(* IEC 61131-3 sources: MotionTestBenchMaster/Logical/02_HMI/0210_PAR/PAR, 10 files *)

(* ---- HMI_PAC_1.st ---- *)
(*HMI_PAC_1 Initialization Action for Filler PLC*)
(*Author = UTERF*)
(*DB Version : 0.11*)
(*File Version : 2.88*)

ACTION HMI_PAC_1_Init :
        HMI_PAC_1._000 := 0;
        HMI_PAC_1._001 := 20;
        HMI_PAC_1._002 := 200;
        HMI_PAC_1._003 := 0;
        HMI_PAC_1._004 := 1;
        HMI_PAC_1._005 := 1;
        HMI_PAC_1._006 := 1;
        HMI_PAC_1._007 := 210;
        HMI_PAC_1._008 := 105;
        HMI_PAC_1._009 := 0;
        HMI_PAC_1._013 := 205;
        HMI_PAC_1._014 := 0;
        HMI_PAC_1._016 := 0;
        HMI_PAC_1._017 := 0;
        HMI_PAC_1._018 := 0;
        HMI_PAC_1._019 := 89;
        HMI_PAC_1._020 := 118;
        HMI_PAC_1._021 := 0;
        HMI_PAC_1._022 := 0;
        HMI_PAC_1._023 := 0;
        HMI_PAC_1._024 := 0;
        HMI_PAC_1._045 := 0;
        HMI_PAC_1._070 := 0;
        HMI_PAC_1._071 := 0;
        HMI_PAC_1._100 := 91;
        HMI_PAC_1._101 := 75;
        HMI_PAC_1._102 := 5;
        HMI_PAC_1._103 := 0;
        HMI_PAC_1._104 := 85;
        HMI_PAC_1._105 := 0;
        HMI_PAC_1._106 := 0;
        HMI_PAC_1._107 := 0;
        HMI_PAC_1._108 := 0;
        HMI_PAC_1._110 := 0;
        HMI_PAC_1._111 := 0;
        HMI_PAC_1._112 := 0;
        HMI_PAC_1._113 := 0;
        HMI_PAC_1._114 := 0;
        HMI_PAC_1._115 := 0;
        HMI_PAC_1._117 := 0;
        HMI_PAC_1._118 := 0;
        HMI_PAC_1._120 := 0;
        HMI_PAC_1._121 := 0;
        HMI_PAC_1._122 := 0;
        HMI_PAC_1._123 := 0;
        HMI_PAC_1._124 := 0;
        HMI_PAC_1._125 := 0;
        HMI_PAC_1._126 := 0;
        HMI_PAC_1._127 := 0;
        HMI_PAC_1._128 := 0;
        HMI_PAC_1._129 := 1;
        HMI_PAC_1._130 := 33;
        HMI_PAC_1._131 := 1;
        HMI_PAC_1._132 := 0;
        HMI_PAC_1._133 := 1;
        HMI_PAC_1._134 := 1;
        HMI_PAC_1._145 := 0;
        HMI_PAC_1._146 := 0;
        HMI_PAC_1._150 := 6;
        HMI_PAC_1._151 := 1;
        HMI_PAC_1._152 := 74;
        HMI_PAC_1._200 := 0;
        HMI_PAC_1._201 := 0;
        HMI_PAC_1._202 := 0;
        HMI_PAC_1._203 := 0;
        HMI_PAC_1._204 := 0;
        HMI_PAC_1._205 := 0;
        HMI_PAC_1._206 := 0;
        HMI_PAC_1._207 := 0;
        HMI_PAC_1._208 := 0;
        HMI_PAC_1._209 := 0;
        HMI_PAC_1._210 := 0;
        HMI_PAC_1._211 := 0;
        HMI_PAC_1._212 := 0;
        HMI_PAC_1._213 := 0;
        HMI_PAC_1._214 := 0;
        HMI_PAC_1._215 := 0;
        HMI_PAC_1._219 := 0;
        HMI_PAC_1._220 := 0;
        HMI_PAC_1._245 := 0;
        HMI_PAC_1._246 := 0;
        HMI_PAC_1._300 := 0;
        HMI_PAC_1._301 := 0;
        HMI_PAC_1._302 := 0;
        HMI_PAC_1._303 := 0;
        HMI_PAC_1._304 := 0;
        HMI_PAC_1._305 := 0;
        HMI_PAC_1._306 := 0;
        HMI_PAC_1._307 := 0;
        HMI_PAC_1._400 := 0;
        HMI_PAC_1._401 := 0;
        HMI_PAC_1._402 := 0;
        HMI_PAC_1._403 := 0;
        HMI_PAC_1._404 := 0;
        HMI_PAC_1._405 := 0;
        HMI_PAC_1._406 := 0;
        HMI_PAC_1._407 := 0;
        HMI_PAC_1._408 := 0;
        HMI_PAC_1._409 := 0;
        HMI_PAC_1._410 := 0;
        HMI_PAC_1._411 := 0;
        HMI_PAC_1._412 := 0;
        HMI_PAC_1._413 := 0;
        HMI_PAC_1._415 := 0;
        HMI_PAC_1._416 := 0;
        HMI_PAC_1._417 := 0;
        HMI_PAC_1._418 := 0;
        HMI_PAC_1._419 := 0;
        HMI_PAC_1._420 := 0;
        HMI_PAC_1._422 := 0;
        HMI_PAC_1._423 := 0;
        HMI_PAC_1._500 := 0;
        HMI_PAC_1._501 := 0;
        HMI_PAC_1._502 := 0;
        HMI_PAC_1._503 := 0;
        HMI_PAC_1._504 := 0;
        HMI_PAC_1._510 := 0;
        HMI_PAC_1._600 := 0;
        HMI_PAC_1._601 := 0;
        HMI_PAC_1._605 := 0;
        HMI_PAC_1._606 := 0;
        HMI_PAC_1._610 := 0;
        HMI_PAC_1._700 := 0;
        HMI_PAC_1._701 := 0;
        HMI_PAC_1._702 := 0;
        HMI_PAC_1._703 := 0;
        HMI_PAC_1._704 := 1;
        HMI_PAC_1._705 := 1;
        HMI_PAC_1._706 := 1;
        HMI_PAC_1._800 := 0;
END_ACTION

(* ---- HMI_PAM_1.st ---- *)
(*HMI_PAM_1 Initialization Action for Filler PLC*)
(*Author = ????*)
(*DB Version : 0.10*)
(*File Version : 2.88*)

ACTION HMI_PAM_1_Init :
        HMI_PAM_1._000 := 50;
        HMI_PAM_1._001 := 20000;
        HMI_PAM_1._002 := 60;
        HMI_PAM_1._003 := 5000;
        HMI_PAM_1._004 := 8000;
        HMI_PAM_1._005 := 5000;
        HMI_PAM_1._006 := 25000;
        HMI_PAM_1._007 := 15000;
        HMI_PAM_1._008 := 20000;
        HMI_PAM_1._009 := 20000;
        HMI_PAM_1._010 := 1500;
        HMI_PAM_1._011 := 8;
        HMI_PAM_1._012 := 8;
        HMI_PAM_1._013 := 0.13;
        HMI_PAM_1._014 := 20000;
        HMI_PAM_1._015 := 20000;
        HMI_PAM_1._020 := 55200;
        HMI_PAM_1._021 := 400;
        HMI_PAM_1._022 := 2;
        HMI_PAM_1._023 := 600;
        HMI_PAM_1._030 := 300;
        HMI_PAM_1._031 := 2;
        HMI_PAM_1._032 := 2;
        HMI_PAM_1._036 := 0;
        HMI_PAM_1._040 := 300;
        HMI_PAM_1._041 := 5;
        HMI_PAM_1._044 := 0;
        HMI_PAM_1._045 := 0;
        HMI_PAM_1._046 := 0;
        HMI_PAM_1._047 := 0;
        HMI_PAM_1._048 := 10;
        HMI_PAM_1._049 := 1;
        HMI_PAM_1._050 := 60;
        HMI_PAM_1._051 := 0;
        HMI_PAM_1._052 := 0;
        HMI_PAM_1._053 := 0;
        HMI_PAM_1._054 := 0;
        HMI_PAM_1._055 := 10000;
        HMI_PAM_1._056 := 20000;
        HMI_PAM_1._057 := 0;
        HMI_PAM_1._058 := 0;
        HMI_PAM_1._060 := 5;
        HMI_PAM_1._061 := 100;
        HMI_PAM_1._065 := 50;
        HMI_PAM_1._080 := 0;
        HMI_PAM_1._081 := 0;
        HMI_PAM_1._082 := 0;
        HMI_PAM_1._083 := 0;
        HMI_PAM_1._084 := 0;
        HMI_PAM_1._085 := 0;
        HMI_PAM_1._086 := 3;
        HMI_PAM_1._087 := 3;
        HMI_PAM_1._088 := 3;
        HMI_PAM_1._089 := 3;
        HMI_PAM_1._090 := 1000000;
        HMI_PAM_1._091 := 40000;
        HMI_PAM_1._092 := 3.2;
        HMI_PAM_1._093 := 3.2;
        HMI_PAM_1._100 := 0;
        HMI_PAM_1._101 := 0;
        HMI_PAM_1._102 := 0;
        HMI_PAM_1._103 := 100;
        HMI_PAM_1._104 := 100;
        HMI_PAM_1._105 := 2;
        HMI_PAM_1._106 := 15;
        HMI_PAM_1._107 := 10;
        HMI_PAM_1._108 := 5;
        HMI_PAM_1._109 := 5;
        HMI_PAM_1._110 := 25;
        HMI_PAM_1._111 := 15;
        HMI_PAM_1._112 := 30;
        HMI_PAM_1._113 := 20;
        HMI_PAM_1._114 := 2;
        HMI_PAM_1._115 := 30;
        HMI_PAM_1._116 := 10;
        HMI_PAM_1._117 := 20;
        HMI_PAM_1._118 := 30;
        HMI_PAM_1._130 := 0;
        HMI_PAM_1._131 := 0;
        HMI_PAM_1._140 := 0;
        HMI_PAM_1._141 := 0;
        HMI_PAM_1._142 := 0;
        HMI_PAM_1._143 := 0;
        HMI_PAM_1._144 := 0;
        HMI_PAM_1._150 := 0;
        HMI_PAM_1._151 := 0;
        HMI_PAM_1._152 := 0;
        HMI_PAM_1._153 := 0;
        HMI_PAM_1._154 := 0;
        HMI_PAM_1._155 := 0;
        HMI_PAM_1._156 := 0;
        HMI_PAM_1._200 := 0;
        HMI_PAM_1._201 := 0;
        HMI_PAM_1._202 := 0;
        HMI_PAM_1._203 := 0;
        HMI_PAM_1._204 := 0;
        HMI_PAM_1._215 := 200;
        HMI_PAM_1._216 := 100;
        HMI_PAM_1._217 := 0;
        HMI_PAM_1._218 := 0;
        HMI_PAM_1._220 := 0;
        HMI_PAM_1._221 := 0;
        HMI_PAM_1._222 := 0;
        HMI_PAM_1._223 := 0;
        HMI_PAM_1._224 := 0;
        HMI_PAM_1._235 := 100;
        HMI_PAM_1._236 := 50;
        HMI_PAM_1._237 := 0;
        HMI_PAM_1._238 := 0;
        HMI_PAM_1._300 := 50;
        HMI_PAM_1._301 := 60;
        HMI_PAM_1._302 := 80;
        HMI_PAM_1._305 := 50;
        HMI_PAM_1._306 := 60;
        HMI_PAM_1._307 := 80;
        HMI_PAM_1._310 := 50;
        HMI_PAM_1._311 := 60;
        HMI_PAM_1._312 := 80;
        HMI_PAM_1._315 := 60;
        HMI_PAM_1._316 := 65;
        HMI_PAM_1._317 := 80;
        HMI_PAM_1._396 := 0;
        HMI_PAM_1._397 := 0;
        HMI_PAM_1._398 := 0;
        HMI_PAM_1._399 := 0;
        HMI_PAM_1._400 := 220;
        HMI_PAM_1._401 := 40;
        HMI_PAM_1._402 := 10;
        HMI_PAM_1._403 := 1;
        HMI_PAM_1._404 := 96;
        HMI_PAM_1._405 := 276;
        HMI_PAM_1._406 := 0;
        HMI_PAM_1._407 := 1;
        HMI_PAM_1._408 := 0;
        HMI_PAM_1._409 := 0;
        HMI_PAM_1._410 := 0;
        HMI_PAM_1._411 := 0;
        HMI_PAM_1._412 := 0;
        HMI_PAM_1._413 := 0;
        HMI_PAM_1._414 := 0;
        HMI_PAM_1._415 := 0;
        HMI_PAM_1._416 := 0;
        HMI_PAM_1._417 := 0;
        HMI_PAM_1._418 := 0;
        HMI_PAM_1._419 := 0;
        HMI_PAM_1._420 := 0;
        HMI_PAM_1._421 := 0;
        HMI_PAM_1._422 := 0;
        HMI_PAM_1._423 := 0;
        HMI_PAM_1._424 := 0;
        HMI_PAM_1._425 := 0;
        HMI_PAM_1._426 := 0;
        HMI_PAM_1._427 := 0;
        HMI_PAM_1._428 := 0;
        HMI_PAM_1._429 := 0;
        HMI_PAM_1._430 := 0;
        HMI_PAM_1._431 := 0;
        HMI_PAM_1._432 := 0;
        HMI_PAM_1._433 := 0;
        HMI_PAM_1._434 := 0;
        HMI_PAM_1._435 := 0;
        HMI_PAM_1._450 := 0;
        HMI_PAM_1._451 := 0;
        HMI_PAM_1._452 := 0;
        HMI_PAM_1._453 := 0;
        HMI_PAM_1._454 := 0;
        HMI_PAM_1._500 := 5;
        HMI_PAM_1._501 := 5;
        HMI_PAM_1._502 := 5;
        HMI_PAM_1._503 := 5;
        HMI_PAM_1._504 := 5;
        HMI_PAM_1._505 := 5;
        HMI_PAM_1._506 := 5;
        HMI_PAM_1._507 := 5;
        HMI_PAM_1._508 := 5;
        HMI_PAM_1._509 := 5;
        HMI_PAM_1._510 := 5;
        HMI_PAM_1._511 := 5;
        HMI_PAM_1._512 := 5;
        HMI_PAM_1._513 := 5;
        HMI_PAM_1._514 := 5;
        HMI_PAM_1._515 := 5;
        HMI_PAM_1._516 := 5;
        HMI_PAM_1._517 := 5;
        HMI_PAM_1._518 := 5;
        HMI_PAM_1._519 := 5;
        HMI_PAM_1._520 := 5;
        HMI_PAM_1._521 := 5;
        HMI_PAM_1._524 := 5;
        HMI_PAM_1._525 := 5;
        HMI_PAM_1._526 := 5;
        HMI_PAM_1._527 := 5;
        HMI_PAM_1._550 := 30;
        HMI_PAM_1._551 := 10;
        HMI_PAM_1._559 := 0;
        HMI_PAM_1._560 := 1;
        HMI_PAM_1._561 := 0;
        HMI_PAM_1._562 := 1;
END_ACTION

(* ---- HMI_PAM_3.st ---- *)
(*HMI_PAM_3 Initialization Action for Filler PLC*)
(*Author = ????*)
(*DB Version : 0.00*)
(*File Version : 2.88*)

ACTION HMI_PAM_3_Init :
        HMI_PAM_3._000 := 80;
        HMI_PAM_3._010 := 8000;
        HMI_PAM_3._100 := 2500;
        HMI_PAM_3._101 := 2500;
        HMI_PAM_3._102 := 0;
        HMI_PAM_3._103 := 0;
        HMI_PAM_3._104 := 0;
        HMI_PAM_3._105 := 0;
        HMI_PAM_3._106 := 0;
        HMI_PAM_3._107 := 0;
        HMI_PAM_3._108 := 0;
        HMI_PAM_3._109 := 0;
        HMI_PAM_3._112 := 0;
        HMI_PAM_3._113 := 0;
        HMI_PAM_3._400 := 4;
        HMI_PAM_3._401 := 4;
        HMI_PAM_3._410 := 0;
        HMI_PAM_3._500 := 3;
        HMI_PAM_3._501 := 5;
        HMI_PAM_3._502 := 3;
        HMI_PAM_3._503 := 20;
        HMI_PAM_3._504 := 50000;
        HMI_PAM_3._505 := 10;
        HMI_PAM_3._506 := 3;
        HMI_PAM_3._507 := 5;
        HMI_PAM_3._508 := 3;
        HMI_PAM_3._510 := 1;
        HMI_PAM_3._511 := 19295;
        HMI_PAM_3._512 := 131976;
        HMI_PAM_3._513 := 3;
        HMI_PAM_3._520 := 100;
        HMI_PAM_3._521 := 100;
        HMI_PAM_3._525 := 3;
        HMI_PAM_3._526 := 300;
        HMI_PAM_3._527 := 1;
        HMI_PAM_3._528 := 0;
        HMI_PAM_3._529 := 1800;
        HMI_PAM_3._530 := 3;
        HMI_PAM_3._531 := 300;
        HMI_PAM_3._532 := 1;
        HMI_PAM_3._534 := 1800;
        HMI_PAM_3._540 := 0;
        HMI_PAM_3._550 := 0;
        HMI_PAM_3._551 := 100;
        HMI_PAM_3._554 := 0;
        HMI_PAM_3._555 := 100;
        HMI_PAM_3._558 := 0;
        HMI_PAM_3._559 := 100;
        HMI_PAM_3._562 := 0;
        HMI_PAM_3._563 := 100;
        HMI_PAM_3._566 := 0;
        HMI_PAM_3._567 := 60;
        HMI_PAM_3._570 := 0;
        HMI_PAM_3._571 := 65;
        HMI_PAM_3._572 := 0;
        HMI_PAM_3._573 := 65;
        HMI_PAM_3._574 := 0;
        HMI_PAM_3._575 := 65;
        HMI_PAM_3._600 := 0;
        HMI_PAM_3._601 := 0;
        HMI_PAM_3._602 := 0;
        HMI_PAM_3._603 := 0;
        HMI_PAM_3._604 := 0;
        HMI_PAM_3._605 := 0;
        HMI_PAM_3._606 := 0;
        HMI_PAM_3._607 := 0;
        HMI_PAM_3._608 := 0;
        HMI_PAM_3._609 := 0;
        HMI_PAM_3._620 := 0;
        HMI_PAM_3._621 := 0;
        HMI_PAM_3._622 := 0;
        HMI_PAM_3._623 := 0;
        HMI_PAM_3._624 := 0;
        HMI_PAM_3._625 := 0;
        HMI_PAM_3._626 := 0;
        HMI_PAM_3._627 := 0;
        HMI_PAM_3._628 := 0;
        HMI_PAM_3._629 := 0;
        HMI_PAM_3._640 := 0;
        HMI_PAM_3._641 := 0;
        HMI_PAM_3._642 := 0;
        HMI_PAM_3._643 := 0;
        HMI_PAM_3._644 := 0;
END_ACTION

(* ---- HMI_PAM_A1.st ---- *)
(*HMI_PAM_A1 Initialization Action for Filler PLC*)
(*Author = ????*)
(*DB Version : 0.00*)
(*File Version : 2.88*)

ACTION HMI_PAM_A1_Init :
        HMI_PAM_A1._000 := 0;
        HMI_PAM_A1._001 := 0;
        HMI_PAM_A1._002 := 0;
        HMI_PAM_A1._005 := 0;
        HMI_PAM_A1._006 := 0;
        HMI_PAM_A1._007 := 0;
        HMI_PAM_A1._010 := 0;
        HMI_PAM_A1._011 := 0;
        HMI_PAM_A1._012 := 0;
        HMI_PAM_A1._015 := 0;
        HMI_PAM_A1._016 := 0;
        HMI_PAM_A1._017 := 0;
        HMI_PAM_A1._020 := 0;
        HMI_PAM_A1._021 := 0;
        HMI_PAM_A1._022 := 0;
        HMI_PAM_A1._025 := 0;
        HMI_PAM_A1._026 := 0;
        HMI_PAM_A1._027 := 0;
        HMI_PAM_A1._030 := 0;
        HMI_PAM_A1._031 := 0;
        HMI_PAM_A1._032 := 0;
        HMI_PAM_A1._035 := 0;
        HMI_PAM_A1._036 := 0;
        HMI_PAM_A1._037 := 0;
        HMI_PAM_A1._040 := 0;
        HMI_PAM_A1._041 := 0;
        HMI_PAM_A1._042 := 0;
        HMI_PAM_A1._045 := 0;
        HMI_PAM_A1._046 := 0;
        HMI_PAM_A1._047 := 0;
        HMI_PAM_A1._050 := 0;
        HMI_PAM_A1._051 := 0;
        HMI_PAM_A1._052 := 0;
        HMI_PAM_A1._055 := 0;
        HMI_PAM_A1._056 := 0;
        HMI_PAM_A1._057 := 0;
        HMI_PAM_A1._060 := 0;
        HMI_PAM_A1._061 := 0;
        HMI_PAM_A1._062 := 0;
END_ACTION

(* ---- HMI_PAM_B1.st ---- *)
(*HMI_PAM_B1 Initialization Action for Filler PLC*)
(*Author = ????*)
(*DB Version : 0.00*)
(*File Version : 2.88*)

ACTION HMI_PAM_B1_Init :
        HMI_PAM_B1._000 := 0;
        HMI_PAM_B1._001 := 40;
        HMI_PAM_B1._005 := 1;
        HMI_PAM_B1._006 := 40;
        HMI_PAM_B1._010 := 0;
        HMI_PAM_B1._011 := 40;
        HMI_PAM_B1._015 := 1;
        HMI_PAM_B1._016 := 40;
        HMI_PAM_B1._020 := 0;
        HMI_PAM_B1._021 := 40;
        HMI_PAM_B1._025 := 1;
        HMI_PAM_B1._026 := 40;
        HMI_PAM_B1._030 := 0;
        HMI_PAM_B1._031 := 40;
        HMI_PAM_B1._035 := 1;
        HMI_PAM_B1._036 := 40;
        HMI_PAM_B1._040 := 0;
        HMI_PAM_B1._041 := 40;
        HMI_PAM_B1._045 := 1;
        HMI_PAM_B1._046 := 40;
        HMI_PAM_B1._050 := 1;
        HMI_PAM_B1._051 := 40;
        HMI_PAM_B1._500 := 5;
        HMI_PAM_B1._501 := 60;
        HMI_PAM_B1._505 := 0;
        HMI_PAM_B1._506 := 100;
        HMI_PAM_B1._510 := 0;
        HMI_PAM_B1._511 := 100;
        HMI_PAM_B1._515 := 0;
        HMI_PAM_B1._516 := 100;
        HMI_PAM_B1._520 := 0;
        HMI_PAM_B1._521 := 100;
        HMI_PAM_B1._525 := 0;
        HMI_PAM_B1._526 := 100;
        HMI_PAM_B1._530 := 0;
        HMI_PAM_B1._531 := 100;
        HMI_PAM_B1._535 := 0;
        HMI_PAM_B1._536 := 100;
        HMI_PAM_B1._540 := 0;
        HMI_PAM_B1._541 := 100;
        HMI_PAM_B1._545 := 0;
        HMI_PAM_B1._546 := 100;
END_ACTION

(* ---- HMI_PAM_C1.st ---- *)
(*HMI_PAM_C1 Initialization Action for Filler PLC*)
(*Author = ????*)
(*DB Version : 0.00*)
(*File Version : 2.88*)

ACTION HMI_PAM_C1_Init :
        HMI_PAM_C1._000 := 0;
        HMI_PAM_C1._001 := 0;
        HMI_PAM_C1._002 := 0;
        HMI_PAM_C1._003 := 0;
        HMI_PAM_C1._004 := 0;
        HMI_PAM_C1._005 := 0;
        HMI_PAM_C1._006 := 0;
        HMI_PAM_C1._007 := 0;
        HMI_PAM_C1._008 := 0;
        HMI_PAM_C1._009 := 0;
        HMI_PAM_C1._010 := 0;
        HMI_PAM_C1._011 := 0;
        HMI_PAM_C1._012 := 0;
        HMI_PAM_C1._013 := 0;
        HMI_PAM_C1._014 := 0;
        HMI_PAM_C1._015 := 0;
        HMI_PAM_C1._016 := 0;
        HMI_PAM_C1._017 := 0;
        HMI_PAM_C1._018 := 0;
        HMI_PAM_C1._019 := 0;
        HMI_PAM_C1._020 := 0;
        HMI_PAM_C1._021 := 0;
        HMI_PAM_C1._022 := 0;
        HMI_PAM_C1._023 := 0;
        HMI_PAM_C1._024 := 0;
        HMI_PAM_C1._025 := 0;
        HMI_PAM_C1._026 := 0;
        HMI_PAM_C1._027 := 0;
        HMI_PAM_C1._028 := 0;
        HMI_PAM_C1._029 := 0;
        HMI_PAM_C1._030 := 0;
        HMI_PAM_C1._031 := 0;
        HMI_PAM_C1._032 := 0;
        HMI_PAM_C1._033 := 0;
        HMI_PAM_C1._034 := 0;
        HMI_PAM_C1._035 := 0;
        HMI_PAM_C1._036 := 0;
        HMI_PAM_C1._037 := 0;
        HMI_PAM_C1._038 := 0;
        HMI_PAM_C1._039 := 0;
        HMI_PAM_C1._040 := 0;
        HMI_PAM_C1._041 := 0;
        HMI_PAM_C1._042 := 0;
        HMI_PAM_C1._043 := 0;
        HMI_PAM_C1._044 := 0;
        HMI_PAM_C1._045 := 0;
        HMI_PAM_C1._046 := 0;
        HMI_PAM_C1._047 := 0;
        HMI_PAM_C1._048 := 0;
        HMI_PAM_C1._049 := 0;
        HMI_PAM_C1._050 := 0;
        HMI_PAM_C1._051 := 0;
        HMI_PAM_C1._052 := 0;
        HMI_PAM_C1._053 := 0;
        HMI_PAM_C1._054 := 0;
        HMI_PAM_C1._055 := 0;
        HMI_PAM_C1._056 := 0;
        HMI_PAM_C1._057 := 0;
        HMI_PAM_C1._058 := 0;
        HMI_PAM_C1._059 := 0;
        HMI_PAM_C1._060 := 0;
        HMI_PAM_C1._061 := 0;
        HMI_PAM_C1._062 := 0;
        HMI_PAM_C1._063 := 0;
        HMI_PAM_C1._064 := 0;
        HMI_PAM_C1._065 := 0;
        HMI_PAM_C1._066 := 0;
        HMI_PAM_C1._067 := 0;
        HMI_PAM_C1._068 := 0;
        HMI_PAM_C1._069 := 0;
        HMI_PAM_C1._070 := 0;
        HMI_PAM_C1._071 := 0;
        HMI_PAM_C1._072 := 0;
        HMI_PAM_C1._073 := 0;
        HMI_PAM_C1._074 := 0;
        HMI_PAM_C1._075 := 0;
        HMI_PAM_C1._076 := 0;
        HMI_PAM_C1._077 := 0;
        HMI_PAM_C1._078 := 0;
        HMI_PAM_C1._079 := 0;
        HMI_PAM_C1._080 := 0;
        HMI_PAM_C1._081 := 0;
        HMI_PAM_C1._082 := 0;
        HMI_PAM_C1._083 := 0;
        HMI_PAM_C1._084 := 0;
        HMI_PAM_C1._085 := 0;
        HMI_PAM_C1._086 := 0;
        HMI_PAM_C1._087 := 0;
        HMI_PAM_C1._088 := 0;
        HMI_PAM_C1._089 := 0;
        HMI_PAM_C1._090 := 0;
        HMI_PAM_C1._091 := 0;
        HMI_PAM_C1._092 := 0;
        HMI_PAM_C1._093 := 0;
        HMI_PAM_C1._094 := 0;
        HMI_PAM_C1._095 := 0;
        HMI_PAM_C1._096 := 0;
        HMI_PAM_C1._097 := 0;
        HMI_PAM_C1._098 := 0;
        HMI_PAM_C1._099 := 0;
        HMI_PAM_C1._100 := 0;
        HMI_PAM_C1._101 := 0;
        HMI_PAM_C1._102 := 0;
        HMI_PAM_C1._103 := 0;
        HMI_PAM_C1._104 := 0;
        HMI_PAM_C1._105 := 0;
        HMI_PAM_C1._106 := 0;
        HMI_PAM_C1._107 := 0;
        HMI_PAM_C1._108 := 0;
        HMI_PAM_C1._109 := 0;
        HMI_PAM_C1._110 := 0;
        HMI_PAM_C1._111 := 0;
        HMI_PAM_C1._112 := 0;
        HMI_PAM_C1._113 := 0;
        HMI_PAM_C1._114 := 0;
        HMI_PAM_C1._115 := 0;
        HMI_PAM_C1._116 := 0;
        HMI_PAM_C1._117 := 0;
        HMI_PAM_C1._118 := 0;
        HMI_PAM_C1._119 := 0;
END_ACTION

(* ---- HMI_PAM_D1.st ---- *)
(*HMI_PAM_D1 Initialization Action for Filler PLC*)
(*Author = ????*)
(*DB Version : 0.00*)
(*File Version : 2.88*)

ACTION HMI_PAM_D1_Init :
        HMI_PAM_D1._000 := 0;
        HMI_PAM_D1._001 := 0;
        HMI_PAM_D1._002 := 0;
        HMI_PAM_D1._003 := 0;
        HMI_PAM_D1._004 := 0;
        HMI_PAM_D1._005 := 0.5;
        HMI_PAM_D1._006 := 1;
        HMI_PAM_D1._007 := 0;
        HMI_PAM_D1._008 := 0;
        HMI_PAM_D1._009 := 0;
        HMI_PAM_D1._010 := 0;
        HMI_PAM_D1._011 := 0;
        HMI_PAM_D1._012 := 0;
        HMI_PAM_D1._013 := 0;
        HMI_PAM_D1._014 := 0;
        HMI_PAM_D1._015 := 0;
        HMI_PAM_D1._016 := 0;
        HMI_PAM_D1._017 := 0;
        HMI_PAM_D1._018 := 0;
        HMI_PAM_D1._019 := 0;
        HMI_PAM_D1._020 := 0;
        HMI_PAM_D1._021 := 0;
        HMI_PAM_D1._022 := 0;
        HMI_PAM_D1._023 := 0;
        HMI_PAM_D1._024 := 0;
        HMI_PAM_D1._025 := 0;
        HMI_PAM_D1._026 := 0;
        HMI_PAM_D1._027 := 0;
        HMI_PAM_D1._028 := 0;
        HMI_PAM_D1._029 := 0;
        HMI_PAM_D1._030 := 0;
        HMI_PAM_D1._031 := 0;
        HMI_PAM_D1._032 := 0;
        HMI_PAM_D1._033 := 0;
        HMI_PAM_D1._034 := 0;
        HMI_PAM_D1._035 := 0;
        HMI_PAM_D1._036 := 0;
        HMI_PAM_D1._037 := 0;
        HMI_PAM_D1._038 := 0;
        HMI_PAM_D1._039 := 0;
        HMI_PAM_D1._040 := 0;
        HMI_PAM_D1._041 := 0;
        HMI_PAM_D1._042 := 0;
        HMI_PAM_D1._043 := 0;
        HMI_PAM_D1._044 := 0;
        HMI_PAM_D1._045 := 0;
        HMI_PAM_D1._046 := 0;
        HMI_PAM_D1._047 := 0;
        HMI_PAM_D1._048 := 0;
        HMI_PAM_D1._049 := 0;
        HMI_PAM_D1._050 := 0;
        HMI_PAM_D1._051 := 0;
        HMI_PAM_D1._052 := 0;
        HMI_PAM_D1._053 := 0;
        HMI_PAM_D1._054 := 0;
        HMI_PAM_D1._055 := 0;
        HMI_PAM_D1._056 := 0;
        HMI_PAM_D1._057 := 0;
        HMI_PAM_D1._058 := 0;
        HMI_PAM_D1._059 := 0;
        HMI_PAM_D1._060 := 0;
        HMI_PAM_D1._061 := 0;
        HMI_PAM_D1._062 := 0;
        HMI_PAM_D1._063 := 0;
        HMI_PAM_D1._064 := 0;
        HMI_PAM_D1._065 := 0;
        HMI_PAM_D1._066 := 0;
        HMI_PAM_D1._067 := 0;
        HMI_PAM_D1._068 := 0;
        HMI_PAM_D1._069 := 0;
        HMI_PAM_D1._070 := 0;
        HMI_PAM_D1._071 := 0;
        HMI_PAM_D1._072 := 0;
        HMI_PAM_D1._073 := 0;
        HMI_PAM_D1._074 := 0;
        HMI_PAM_D1._075 := 0;
        HMI_PAM_D1._076 := 0;
        HMI_PAM_D1._077 := 0;
        HMI_PAM_D1._078 := 0;
        HMI_PAM_D1._079 := 0;
        HMI_PAM_D1._080 := 0;
        HMI_PAM_D1._081 := 0;
        HMI_PAM_D1._082 := 0;
        HMI_PAM_D1._083 := 0;
        HMI_PAM_D1._084 := 0;
        HMI_PAM_D1._085 := 0;
        HMI_PAM_D1._086 := 0;
        HMI_PAM_D1._087 := 0;
        HMI_PAM_D1._088 := 0;
        HMI_PAM_D1._089 := 0;
        HMI_PAM_D1._090 := 10;
        HMI_PAM_D1._091 := 10;
        HMI_PAM_D1._092 := 1;
        HMI_PAM_D1._093 := 0;
        HMI_PAM_D1._094 := 0;
        HMI_PAM_D1._095 := 0.7;
        HMI_PAM_D1._096 := 1;
        HMI_PAM_D1._097 := 1;
        HMI_PAM_D1._098 := 0;
        HMI_PAM_D1._099 := 0;
        HMI_PAM_D1._500 := 0;
        HMI_PAM_D1._501 := 40;
        HMI_PAM_D1._502 := 0;
        HMI_PAM_D1._503 := 0;
        HMI_PAM_D1._504 := 0;
        HMI_PAM_D1._505 := 1.5;
        HMI_PAM_D1._506 := 0.6;
        HMI_PAM_D1._507 := 0;
        HMI_PAM_D1._508 := 0;
        HMI_PAM_D1._509 := 0;
        HMI_PAM_D1._510 := 0;
        HMI_PAM_D1._511 := 0;
        HMI_PAM_D1._512 := 0;
        HMI_PAM_D1._513 := 0;
        HMI_PAM_D1._514 := 0;
        HMI_PAM_D1._515 := 0;
        HMI_PAM_D1._516 := 0;
        HMI_PAM_D1._517 := 0;
        HMI_PAM_D1._518 := 0;
        HMI_PAM_D1._519 := 0;
        HMI_PAM_D1._520 := 0;
        HMI_PAM_D1._521 := 0;
        HMI_PAM_D1._522 := 0;
        HMI_PAM_D1._523 := 0;
        HMI_PAM_D1._524 := 0;
        HMI_PAM_D1._525 := 0;
        HMI_PAM_D1._526 := 0;
        HMI_PAM_D1._527 := 0;
        HMI_PAM_D1._528 := 0;
        HMI_PAM_D1._529 := 0;
        HMI_PAM_D1._530 := 0;
        HMI_PAM_D1._531 := 0;
        HMI_PAM_D1._532 := 0;
        HMI_PAM_D1._533 := 0;
        HMI_PAM_D1._534 := 0;
        HMI_PAM_D1._535 := 0;
        HMI_PAM_D1._536 := 0;
        HMI_PAM_D1._537 := 0;
        HMI_PAM_D1._538 := 0;
        HMI_PAM_D1._539 := 0;
        HMI_PAM_D1._540 := 0;
        HMI_PAM_D1._541 := 0;
        HMI_PAM_D1._542 := 0;
        HMI_PAM_D1._543 := 0;
        HMI_PAM_D1._544 := 0;
        HMI_PAM_D1._545 := 0;
        HMI_PAM_D1._546 := 0;
        HMI_PAM_D1._547 := 0;
        HMI_PAM_D1._548 := 0;
        HMI_PAM_D1._549 := 0;
        HMI_PAM_D1._550 := 0;
        HMI_PAM_D1._551 := 0;
        HMI_PAM_D1._552 := 0;
        HMI_PAM_D1._553 := 0;
        HMI_PAM_D1._554 := 0;
        HMI_PAM_D1._555 := 0;
        HMI_PAM_D1._556 := 0;
        HMI_PAM_D1._557 := 0;
        HMI_PAM_D1._558 := 0;
        HMI_PAM_D1._559 := 0;
        HMI_PAM_D1._560 := 0;
        HMI_PAM_D1._561 := 0;
        HMI_PAM_D1._562 := 0;
        HMI_PAM_D1._563 := 0;
        HMI_PAM_D1._564 := 0;
        HMI_PAM_D1._565 := 0;
        HMI_PAM_D1._566 := 0;
        HMI_PAM_D1._567 := 0;
        HMI_PAM_D1._568 := 0;
        HMI_PAM_D1._569 := 0;
        HMI_PAM_D1._570 := 0;
        HMI_PAM_D1._571 := 0;
        HMI_PAM_D1._572 := 0;
        HMI_PAM_D1._573 := 0;
        HMI_PAM_D1._574 := 0;
        HMI_PAM_D1._575 := 0;
        HMI_PAM_D1._576 := 0;
        HMI_PAM_D1._577 := 0;
        HMI_PAM_D1._578 := 0;
        HMI_PAM_D1._579 := 0;
        HMI_PAM_D1._580 := 0;
        HMI_PAM_D1._581 := 0;
        HMI_PAM_D1._582 := 0;
        HMI_PAM_D1._583 := 0;
        HMI_PAM_D1._584 := 0;
        HMI_PAM_D1._585 := 0;
        HMI_PAM_D1._586 := 0;
        HMI_PAM_D1._587 := 0;
        HMI_PAM_D1._588 := 0;
        HMI_PAM_D1._589 := 0;
        HMI_PAM_D1._590 := 0;
        HMI_PAM_D1._591 := 0;
        HMI_PAM_D1._592 := 0;
        HMI_PAM_D1._593 := 0;
        HMI_PAM_D1._594 := 0;
        HMI_PAM_D1._595 := 0;
        HMI_PAM_D1._596 := 0;
        HMI_PAM_D1._597 := 0;
        HMI_PAM_D1._598 := 0;
        HMI_PAM_D1._599 := 0;
END_ACTION

(* ---- HMI_PAT_1.st ---- *)
(*HMI_PAT_1 Initialization Action for Filler PLC*)
(*Author = ????*)
(*DB Version : 0.00*)
(*File Version : 2.88*)

ACTION HMI_PAT_1_Init :
        HMI_PAT_1._010 := 0;
        HMI_PAT_1._011 := 0;
        HMI_PAT_1._100 := 150;
        HMI_PAT_1._101 := 200;
        HMI_PAT_1._110 := 20;
        HMI_PAT_1._420 := 450;
        HMI_PAT_1._421 := 1000;
        HMI_PAT_1._422 := 200;
        HMI_PAT_1._423 := 7200;
        HMI_PAT_1._424 := 1800;
        HMI_PAT_1._425 := 20;
        HMI_PAT_1._426 := 600;
END_ACTION

(* ---- PAR.st ---- *)
PROGRAM _INIT
//Call all the option parameters
	HMI_PAO_2;

	//Call all the parameters structure for HMI (RCP excluded)
	HMI_PAC_1;
	HMI_PAM_1;
	HMI_PAM_3;
	HMI_PAM_A1;
	HMI_PAM_B1;
	HMI_PAM_C1;
	HMI_PAM_D1;
	HMI_PAT_1;

	//Call all the parameters configuration structure for HMI (RCP excluded)
	HMI_CFG_PAC_1;
	HMI_CFG_PAM_1;
	HMI_CFG_PAM_3;
	HMI_CFG_PAM_A1;
	HMI_CFG_PAM_B1;
	HMI_CFG_PAM_C1;
	HMI_CFG_PAM_D1;
	HMI_CFG_PAT_1;
END_PROGRAM

PROGRAM _CYCLIC
	HMI_PB[PB_PAR_Initialization].Visibility	:= TRUE;
	HMI_PB[PB_PAR_Initialization].Enable		:= TRUE;

	IF VAR_PAR_Initialization THEN
		HMI_PAC_1_Init;
		HMI_PAM_1_Init;
		HMI_PAM_3_Init;
		HMI_PAM_A1_Init;
		HMI_PAM_B1_Init;
		HMI_PAM_C1_Init;
		HMI_PAM_D1_Init;
		HMI_PAT_1_Init;
		VAR_PAR_Initialization	:= FALSE;
	END_IF

	TMR_TON_ParInitialization(IN	:= HMI_PB[PB_PAR_Initialization].ON,
								PT := t#5s);

	IF CFG_Par.Process.BlendFill THEN
		FlrCrb.HMI_ParInitialization	:= HMI_PB[PB_PAR_Initialization].ON;
	ELSIF CFG_Par.Process.InternalSkid THEN
		FlrSkd.HMI_ParInitialization	:= HMI_PB[PB_PAR_Initialization].ON;
	END_IF

	IF TMR_TON_ParInitialization.Q THEN
		VAR_PAR_Initialization			:= TRUE;
	END_IF

	HMI_PB[PB_PAR_Initialization].Blink		:= HMI_PB[PB_PAR_Initialization].ON AND NOT TMR_TON_ParInitialization.Q;
	HMI_PB[PB_PAR_Initialization].LampON	:= VAR_PAR_Initialization OR TMR_TON_ParInitialization.Q;
END_PROGRAM

(* ---- Variable.var ---- *)
VAR
	TMR_TON_ParInitialization : TON;
	VAR_PAR_Initialization : BOOL;
END_VAR
